(* CODESYS project MID_CAN_Demo.project

Project tree, tasks and I/O mapping:
  Device : Changsha Xiangji-ARM Cortex A9(xilinx zynq7000)-linux, Changsha Xiangji Hiden Technology Co.Ltd, version 3.5.10.20
    application Application
      libraries: Standard, * (System); CAA Callback Extern, * (CAA Technical Workgroup); CAA Can Low Level Extern, * (CAA Technical Workgroup); CAA Can Low Level Imp Extern, * (CAA Technical Workgroup); CAA Types Extern, * (CAA Technical Workgroup); CAN API, 1.0.0.3 (3S - Smart Software Solutions GmbH); SysMem, * (System); VisuDialogs, * (System)
      task MainTask (cyclic, interval 4 ms, priority 1) calls PLC_PRG
      task VISU_TASK (cyclic, interval 100 ms, priority 31) calls VisuElems.Visu_Prg
      program PLC_PRG [ST]
      global variables GVL
      CAN_COMM/
        function CAN_Send_MSG [ST]
      image pool ImagePool
      visualisation Can_Demo_Visua
    SoftMotion General Axis Pool
  5ce3da45-db07-42e7-a21c-a00fff4ed8f6|companyLOG.jpg
  text list GlobalTextList
*)

// Device/Application/GVL
{attribute 'qualified_only'}
{attribute 'qualified_only'}


VAR_GLOBAL
	
	hCan:CAA.HANDLE:=0;
    CanWriteData : ARRAY[0..7] OF BYTE:=[1,2,3,4,5,6,7,8];
    CanWriteMsgID:UDINT:=0;
	CanReadData : ARRAY[0..7] OF BYTE;  
	CanReadMsgID:UDINT;
	
	hCan1:CAA.HANDLE:=0;
    CanWriteMsgID1:UDINT:=1;
	CanWriteData1 : ARRAY[0..7] OF BYTE:=[8,7,6,5,4,3,2,1];
	CanReadMsgID1:UDINT; 
	CanReadData1 : ARRAY[0..7] OF BYTE;  	
	
	

	
END_VAR

// Device/Application/PLC_PRG
PROGRAM PLC_PRG
VAR
		bCanInit:BOOL:=FALSE;	
	bCanInit1:BOOL:=FALSE;	
	hReceiver:CAA.HANDLE;
	hReceiver1:CAA.HANDLE;
	Err:CAA.ERROR;
	Err1:CAA.ERROR;

	
	hMsg : CAA.HANDLE;
	nReceived : CAA.COUNT;
	nAvailable: CAA.COUNT;
	ReadErr   : CAA.ERROR;
	MsgID     : CL2I.COBID;	
	pRxData :POINTER TO CL2I.DATA;
	
	hMsg1 : CAA.HANDLE;
	nReceived1 : CAA.COUNT;
	nAvailable1: CAA.COUNT;
	ReadErr1   : CAA.ERROR;
	MsgID1     : CL2I.COBID;	
	pRxData1 :POINTER TO CL2I.DATA;	
	

END_VAR

//CAN0 接收
IF NOT bCanInit THEN
	GVL.hCan := cl2.DriverOpenH(usiNetId:=0,uiBaudRate:=125,xSupport29Bits:=TRUE,ctMessages:=100,peError:=ADR(Err));	
	
	hReceiver := cl2.CreateMaskReceiver(hDriver := GVL.hCan,
						   cobIdValue := 16#1C1F1D01, 
						   cobIdMask := 16#00000000, 
						   xRTRValue := FALSE, 
                           xRTRMask := TRUE,
						   x29BitIdValue := TRUE, //true接收扩展帧，false接受标准帧
                           x29BitIdMask := FALSE, //false同时接收标准帧和扩展帧，true只接收一种
                           xTransmitValue := FALSE,
                           xTransmitMask := TRUE,
						   xAlwaysNewest := FALSE, 
                           eEvent := CB.EVENT.NO_EVENT, 
                           xEnableSyncWindow := FALSE, 
                           peError := ADR(ReadErr));
END_IF

IF (GVL.hCan <> 0 AND hReceiver <> 0 ) THEN
	 bCanInit := TRUE;
ELSE
	RETURN;
END_IF

nReceived := cl2.GetMsgCount(hReceiverId :=hReceiver, peError := ADR(ReadErr));
IF nReceived <> 0 THEN
	REPEAT
		hMsg := cl2.Read(hReceiverId :=hReceiver,pctMsgLeft:=ADR(nAvailable),peError:=ADR(ReadErr));
		MsgID:= cl2.GetMessageId(hMessage:=hMsg,peError:=ADR(ReadErr));
		pRxData := cl2.GetMessageDataPointer(hMessage:= hMsg,peError:=ADR(ReadErr));	
        SysMemCpy(pDest:=ADR(GVL.CanReadData),pSrc:=pRxData,udiCount:=SIZEOF(GVL.CanReadData));	
		GVL.CanReadMsgID := MsgID;
		cl2.FreeMessage(hMsg);
		
	UNTIL 0=nAvailable
	END_REPEAT
END_IF

//CAN1接收
IF NOT bCanInit1 THEN
	GVL.hCan1 := cl2.DriverOpenH(usiNetId:=1,uiBaudRate:=125,xSupport29Bits:=TRUE,ctMessages:=100,peError:=ADR(Err));	
	
	hReceiver1 := cl2.CreateMaskReceiver(hDriver := GVL.hCan1,
						   cobIdValue := 16#1C1F1D01, 
						   cobIdMask := 16#00000000, 
						   xRTRValue := FALSE, 
                           xRTRMask := TRUE,
						   x29BitIdValue := TRUE, //true接收扩展帧，false接受标准帧
                           x29BitIdMask := FALSE, //false同时接收标准帧和扩展帧，true只接收一种
                           xTransmitValue := FALSE,
                           xTransmitMask := TRUE,
						   xAlwaysNewest := FALSE, 
                           eEvent := CB.EVENT.NO_EVENT, 
                           xEnableSyncWindow := FALSE, 
                           peError := ADR(ReadErr1));
END_IF

IF (GVL.hCan1 <> 0 AND hReceiver1 <> 0 ) THEN
	 bCanInit1 := TRUE;
ELSE
	RETURN;
END_IF

nReceived1 := cl2.GetMsgCount(hReceiverId :=hReceiver1, peError := ADR(ReadErr1));
IF nReceived1 <> 0 THEN
	REPEAT
		hMsg1 := cl2.Read(hReceiverId :=hReceiver1,pctMsgLeft:=ADR(nAvailable1),peError:=ADR(ReadErr1));
		MsgID1:= cl2.GetMessageId(hMessage:=hMsg1,peError:=ADR(ReadErr1));
		pRxData1 := cl2.GetMessageDataPointer(hMessage:= hMsg1,peError:=ADR(ReadErr1));	
        SysMemCpy(pDest:=ADR(GVL.CanReadData1),pSrc:=pRxData1,udiCount:=SIZEOF(GVL.CanReadData1));	
		GVL.CanReadMsgID1 := MsgID1;
		cl2.FreeMessage(hMsg1);
		
	UNTIL 0=nAvailable1
	END_REPEAT
END_IF

END_PROGRAM

// Device/Application/CAN_COMM/CAN_Send_MSG
FUNCTION CAN_Send_MSG : BOOL
VAR_INPUT
	hCan:CAA.HANDLE;	
    TMsgID   : CL2I.COBID;
    TusiLen  : USINT;
	TData    : ARRAY[0..7] OF BYTE;    	
END_VAR
VAR
   Send:CAA.HANDLE;
   WriteErr   : CL2.ERROR;
   p_data:POINTER TO CL2I.DATA;
END_VAR

IF  (0=hCan) THEN
	RETURN;
END_IF 

Send := cl2.CreateMessage(hDriver := hCan,
                          cobID := TMsgID,
						  usiLength := TusiLen,
						  xRTR := FALSE,
						  x29BitID := FALSE,
						  peError := ADR(WriteErr));
						  
IF Send <> CAA.gc_hINVALID THEN
	p_data := cl2.GetMessageDataPointer(hMessage := Send,peError:=ADR(WriteErr));
	IF (WriteErr = CL2.ERROR.NO_ERROR) THEN
		SysMemCpy(pDest:=p_data,pSrc:=ADR(TData),udiCount:=SIZEOF(TData));
	END_IF
	
	WriteErr := cl2.Write(hDriver := hCan,hMessage:=Send,usiPriority:=1,xEnableSyncWindow:=FALSE);
	IF (WriteErr <> CL2.ERROR.NO_ERROR) THEN
        cl2.FreeMessage(hMessage:=Send);		
	END_IF
	
	p_data := CAA.gc_pNULL;
	Send:=CAA.gc_hINVALID;	
END_IF

END_FUNCTION

// Device/Application/Can_Demo_Visua
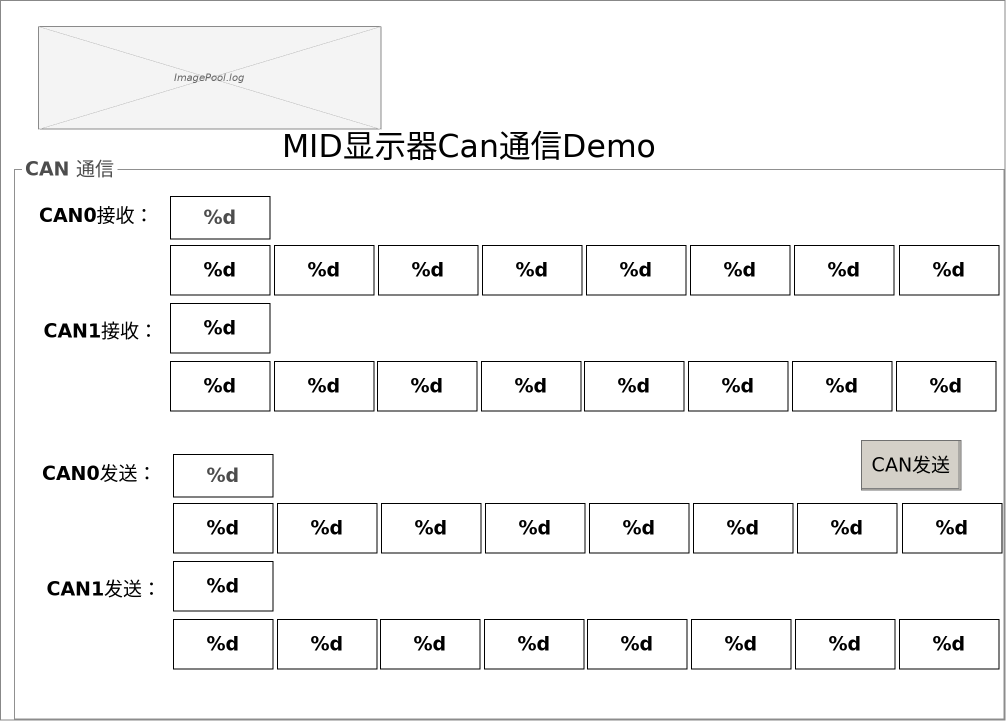
VISUALIZATION Can_Demo_Visua  // 1006x721
    Image (38,26 343x103), image: ImagePool.log
    Label (182,103 574x86), "MID显示器Can通信Demo"
    GroupBox (14,161 990x558), "CAN 通信"
        Label (-4,23 173x63), "CAN0接收："
        Rectangle (156,35 100x43), "%d", text variable: GVL.CanReadMsgID
        Rectangle (885,84 100x50), "%d", text variable: GVL.CanReadData[7]
        Rectangle (780,84 100x50), "%d", text variable: GVL.CanReadData[6]
        Rectangle (676,84 100x50), "%d", text variable: GVL.CanReadData[5]
        Rectangle (572,84 100x50), "%d", text variable: GVL.CanReadData[4]
        Rectangle (468,84 100x50), "%d", text variable: GVL.CanReadData[3]
        Rectangle (364,84 100x50), "%d", text variable: GVL.CanReadData[2]
        Rectangle (260,84 100x50), "%d", text variable: GVL.CanReadData[1]
        Label (11,145 152x50), "CAN1接收："
        Rectangle (156,142 100x50), "%d", text variable: GVL.CanReadMsgID1
            OnMouseDown: write the text variable via VisuDialogs.Numpad, min 0, max 4095
        Rectangle (882,200 100x50), "%d", text variable: GVL.CanReadData1[7]
            OnMouseDown: write the text variable via VisuDialogs.Numpad, min 0, max 255
        Rectangle (778,200 100x50), "%d", text variable: GVL.CanReadData1[6]
            OnMouseDown: write the text variable via VisuDialogs.Numpad, min 0, max 255
        Rectangle (674,200 100x50), "%d", text variable: GVL.CanReadData1[5]
            OnMouseDown: write the text variable via VisuDialogs.Numpad, min 0, max 255
        Rectangle (570,200 100x50), "%d", text variable: GVL.CanReadData1[4]
            OnMouseDown: write the text variable via VisuDialogs.Numpad, min 0, max 255
        Rectangle (467,200 100x50), "%d", text variable: GVL.CanReadData1[3]
            OnMouseDown: write the text variable via VisuDialogs.Numpad, min 0, max 255
        Rectangle (363,200 100x50), "%d", text variable: GVL.CanReadData1[2]
            OnMouseDown: write the text variable via VisuDialogs.Numpad, min 0, max 255
        Rectangle (260,200 100x50), "%d", text variable: GVL.CanReadData1[1]
            OnMouseDown: write the text variable via VisuDialogs.Numpad, min 0, max 255
        Rectangle (156,200 100x50), "%d", text variable: GVL.CanReadData1[0]
            OnMouseDown: write the text variable via VisuDialogs.Numpad, min 0, max 255
        Label (-1,281 173x63), "CAN0发送："
    Rectangle (170,245 100x50), "%d", text variable: GVL.CanReadData[0]
    Rectangle (173,454 100x43), "%d", text variable: GVL.CanWriteMsgID
        OnMouseDown: write the text variable via VisuDialogs.Numpad
    Rectangle (902,503 100x50), "%d", text variable: GVL.CanWriteData[7]
        OnMouseClick: write the text variable via VisuDialogs.Numpad
    Rectangle (797,503 100x50), "%d", text variable: GVL.CanWriteData[6]
        OnMouseClick: write the text variable via VisuDialogs.Numpad
    Rectangle (693,503 100x50), "%d", text variable: GVL.CanWriteData[5]
        OnMouseClick: write the text variable via VisuDialogs.Numpad
    Rectangle (589,503 100x50), "%d", text variable: GVL.CanWriteData[4]
        OnMouseClick: write the text variable via VisuDialogs.Numpad
    Rectangle (485,503 100x50), "%d", text variable: GVL.CanWriteData[3]
        OnMouseClick: write the text variable via VisuDialogs.Numpad
    Rectangle (381,503 100x50), "%d", text variable: GVL.CanWriteData[2]
        OnMouseClick: write the text variable via VisuDialogs.Numpad
    Rectangle (277,503 100x50), "%d", text variable: GVL.CanWriteData[1]
        OnMouseClick: write the text variable via VisuDialogs.Numpad
    Label (28,564 152x50), "CAN1发送："
    Rectangle (173,561 100x50), "%d", text variable: GVL.CanWriteMsgID1
        OnMouseDown: write the text variable via VisuDialogs.Numpad, min 0, max 4095
    Rectangle (899,619 100x50), "%d", text variable: GVL.CanWriteData1[7]
        OnMouseDown: write the text variable via VisuDialogs.Numpad, min 0, max 255
    Rectangle (795,619 100x50), "%d", text variable: GVL.CanWriteData1[6]
        OnMouseDown: write the text variable via VisuDialogs.Numpad, min 0, max 255
    Rectangle (691,619 100x50), "%d", text variable: GVL.CanWriteData1[5]
        OnMouseDown: write the text variable via VisuDialogs.Numpad, min 0, max 255
    Rectangle (587,619 100x50), "%d", text variable: GVL.CanWriteData1[4]
        OnMouseDown: write the text variable via VisuDialogs.Numpad, min 0, max 255
    Rectangle (484,619 100x50), "%d", text variable: GVL.CanWriteData1[3]
        OnMouseDown: write the text variable via VisuDialogs.Numpad, min 0, max 255
    Rectangle (380,619 100x50), "%d", text variable: GVL.CanWriteData1[2]
        OnMouseDown: write the text variable via VisuDialogs.Numpad, min 0, max 255
    Rectangle (277,619 100x50), "%d", text variable: GVL.CanWriteData1[1]
        OnMouseDown: write the text variable via VisuDialogs.Numpad, min 0, max 255
    Rectangle (173,619 100x50), "%d", text variable: GVL.CanWriteData1[0]
        OnMouseDown: write the text variable via VisuDialogs.Numpad, min 0, max 255
    Button (861,440 100x50), "CAN发送"
        OnMouseDown: execute {
            //CAN_Send_MSG(gvl.CanWriteMsgID,8,gvl.CanWriteData);
            (*gvl.CanWriteMsgID:=0;
            gvl.CanWriteData[0]:=1;
            gvl.CanWriteData[1]:=2;
            gvl.CanWriteData[2]:=3;
            gvl.CanWriteData[3]:=4;
            gvl.CanWriteData[4]:=5;
            gvl.CanWriteData[5]:=6;
            gvl.CanWriteData[6]:=7;
            gvl.CanWriteData[7]:=8;
            gvl.CanWriteMsgID1:=1;
            gvl.CanWriteData1[0]:=8;
            gvl.CanWriteData1[1]:=7;
            gvl.CanWriteData1[2]:=6;
            gvl.CanWriteData1[3]:=5;
            gvl.CanWriteData1[4]:=4;
            gvl.CanWriteData1[5]:=3;
            gvl.CanWriteData1[6]:=2;
            gvl.CanWriteData1[7]:=1;*)
            CAN_Send_MSG(GVL.hCan,gvl.CanWriteMsgID,8,gvl.CanWriteData);
            CAN_Send_MSG(GVL.hCan1,gvl.CanWriteMsgID1,8,gvl.CanWriteData1);
        }
    Rectangle (173,503 100x50), "%d", text variable: GVL.CanWriteData[0]
        OnMouseClick: write the text variable via VisuDialogs.Numpad
END_VISUALIZATION
